FUNCTION_BLOCK ElectricBox
VAR_INPUT
END_VAR
VAR_OUTPUT
END_VAR
VAR
END_VAR

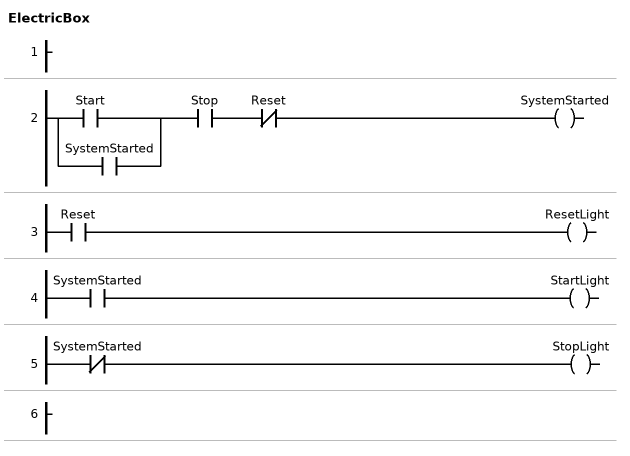
// NETWORK 1

// NETWORK 2
SystemStarted := (Start OR SystemStarted) AND Stop AND NOT Reset;

// NETWORK 3
ResetLight := Reset;

// NETWORK 4
StartLight := SystemStarted;

// NETWORK 5
StopLight := NOT SystemStarted;

// NETWORK 6

END_FUNCTION_BLOCK

(* stored: Version 1.1.0.1, ProductVersion 3.1.4024.6
   POU ElectricBox: Id {66237825-df41-4218-87f0-4073ab762324}, SpecialFunc None *)
